RoboDK station: 新建工作站 (1).rdk

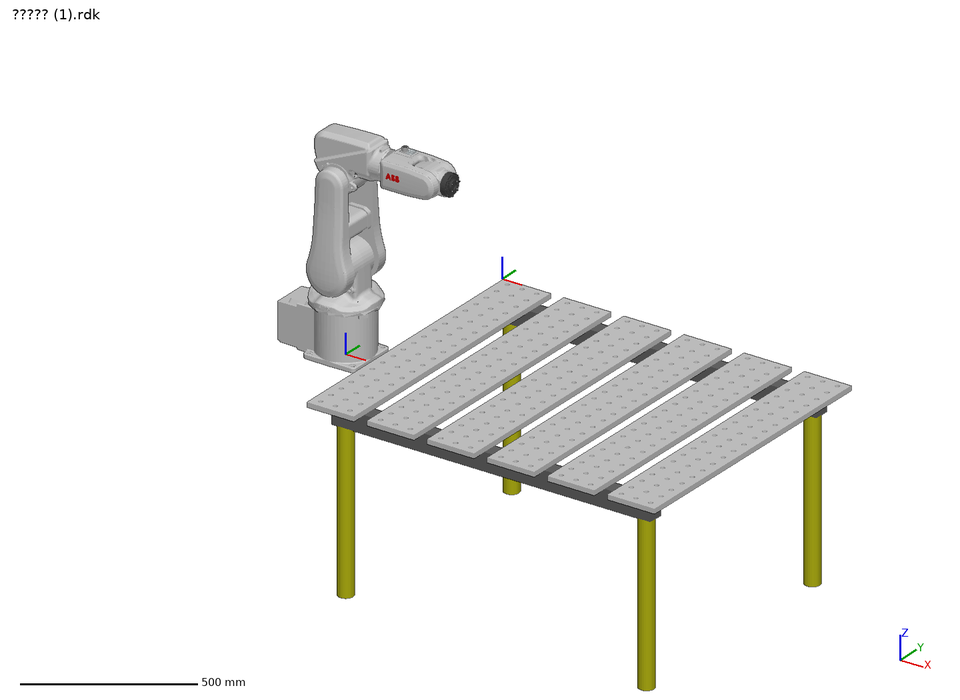
[picture v0: the station drawn from its stored meshes, robots at their saved joint values, targets as dots, program paths as lines]
Station 新建工作站 (1) (saved by RoboDK 5.3.4). Poses are relative to the parent item; angles as X-Y-Z fixed-axis rotations.
  - frame ABB IRB 120-3/0.6 Base at (0, 0, 0) mm
    - robot ABB IRB 120-3/0.6: 6 axes, payload 3 kg, reach 580 mm, repeatability 0.01 mm, weight 25 kg
        modified DH rows (alpha deg, a mm, theta deg, d mm): 0, 0, 0, 290; -90, 0, -90, 0; 0, 270, 0, 0; -90, 70, 0, 302; 90, 0, 0, 0; -90, 0, 180, 72
        joint limits [-165, -110, -90, -160, -120, -400] to [165, 110, 70, 160, 120, 400]; home [0, 0, 0, 0, 0, 0]; saved at [0, 0, 0, 0, 0, 0]
  - object Table at (800, 0, 100) mm, size 1193.8 x 965.2 x 609.6 mm, geometry from welding_table.sld
  - frame worktable at (200, 480, 100) mm
